(* PLC project TankLevelControl, PLCAutoPilot Tank Level Control 1.0 *)
(* stored: creationDateTime 2025-12-25T12:00:00, modificationDateTime 2025-12-25T12:00:00 *)

(* Dual Tank Level Control Program - Controls two pumps for tank filling - Pump 1: Fills Tank 1 from source - Pump 2: Transfers from Tank 1 to RO Tank - Includes start/stop, fault detection, and alarms *)
PROGRAM Tank_Control
  VAR
    System_Running : BOOL := FALSE;  (* System running flag *)
    Pump1_Cmd : BOOL := FALSE;  (* Pump 1 run command *)
    Pump2_Cmd : BOOL := FALSE;  (* Pump 2 run command *)
    Fault_Flag : BOOL := FALSE;  (* Fault active flag *)
    Pump1_Timer : TON;  (* Pump 1 delay timer *)
    Pump2_Timer : TON;  (* Pump 2 delay timer *)
  END_VAR
  VAR_INPUT
    LS_Tank1 : BOOL;  (* Tank 1 Level Switch (0=Low, 1=High) *)
    LS_RO_Tank : BOOL;  (* RO Tank Level Switch (0=Low, 1=High) *)
    PB_Start : BOOL;  (* Start Push Button (NO) *)
    PB_Stop : BOOL;  (* Stop Push Button (NC - TRUE when not pressed) *)
    PB_EStop : BOOL;  (* Emergency Stop (NC - TRUE when not pressed) *)
    OL_Pump1 : BOOL;  (* Pump 1 Overload (NC - TRUE when OK) *)
    OL_Pump2 : BOOL;  (* Pump 2 Overload (NC - TRUE when OK) *)
  END_VAR
  VAR_OUTPUT
    Pump1_Out : BOOL;  (* Pump 1 Output *)
    Pump2_Out : BOOL;  (* Pump 2 Output *)
    Running_Light : BOOL;  (* System Running Indicator *)
    Tank1_Low_Alarm : BOOL;  (* Tank 1 Low Level Alarm *)
    RO_Low_Alarm : BOOL;  (* RO Tank Low Level Alarm *)
    Fault_Light : BOOL;  (* Fault Indicator *)
  END_VAR

            
(* ================================================ *)
(* TANK LEVEL CONTROL PROGRAM                       *)
(* Dual Tank System with Pump Control               *)
(* Generated by PLCAutoPilot                        *)
(* ================================================ *)

(* ----- SYSTEM START/STOP LOGIC ----- *)
(* Start system when Start button pressed and safety OK *)
IF PB_Start AND PB_Stop AND PB_EStop AND NOT Fault_Flag THEN
    System_Running := TRUE;
END_IF;

(* Stop system when Stop button or E-Stop pressed *)
IF NOT PB_Stop OR NOT PB_EStop THEN
    System_Running := FALSE;
END_IF;

(* ----- FAULT DETECTION ----- *)
(* Set fault if any overload trips *)
IF NOT OL_Pump1 OR NOT OL_Pump2 THEN
    Fault_Flag := TRUE;
END_IF;

(* Reset fault when Start pressed and overloads OK *)
IF PB_Start AND OL_Pump1 AND OL_Pump2 THEN
    Fault_Flag := FALSE;
END_IF;

(* ----- PUMP 1 CONTROL (Fill Tank 1) ----- *)
(* Run Pump 1 when system running, Tank 1 is LOW, no fault *)
Pump1_Cmd := System_Running AND NOT LS_Tank1 AND OL_Pump1 AND NOT Fault_Flag;

(* Timer for Pump 1 start delay *)
Pump1_Timer(IN := Pump1_Cmd, PT := T#2S);

(* Pump 1 output with delay *)
Pump1_Out := Pump1_Timer.Q;

(* ----- PUMP 2 CONTROL (Fill RO Tank) ----- *)
(* Run Pump 2 when system running, RO Tank is LOW, Tank 1 is HIGH, no fault *)
Pump2_Cmd := System_Running AND NOT LS_RO_Tank AND LS_Tank1 AND OL_Pump2 AND NOT Fault_Flag;

(* Timer for Pump 2 start delay *)
Pump2_Timer(IN := Pump2_Cmd, PT := T#2S);

(* Pump 2 output with delay *)
Pump2_Out := Pump2_Timer.Q;

(* ----- INDICATOR OUTPUTS ----- *)
Running_Light := System_Running;
Tank1_Low_Alarm := System_Running AND NOT LS_Tank1;
RO_Low_Alarm := System_Running AND NOT LS_RO_Tank;
Fault_Light := Fault_Flag;
            
          
END_PROGRAM

FUNCTION_BLOCK GVL_IO
  VAR
    DI_Tank1_Level AT %IX0.0 : BOOL;  (* Tank 1 Level Switch Input *)
    DI_RO_Tank_Level AT %IX0.1 : BOOL;  (* RO Tank Level Switch Input *)
    DI_Start AT %IX0.2 : BOOL;  (* Start Button Input *)
    DI_Stop AT %IX0.3 : BOOL;  (* Stop Button Input *)
    DI_EStop AT %IX0.4 : BOOL;  (* Emergency Stop Input *)
    DI_OL_Pump1 AT %IX0.5 : BOOL;  (* Pump 1 Overload Input *)
    DI_OL_Pump2 AT %IX0.6 : BOOL;  (* Pump 2 Overload Input *)
    DO_Pump1 AT %QX0.0 : BOOL;  (* Pump 1 Output *)
    DO_Pump2 AT %QX0.1 : BOOL;  (* Pump 2 Output *)
    DO_Running AT %QX0.2 : BOOL;  (* Running Light Output *)
    DO_Tank1_Alarm AT %QX0.3 : BOOL;  (* Tank 1 Low Alarm Output *)
    DO_RO_Alarm AT %QX0.4 : BOOL;  (* RO Tank Low Alarm Output *)
    DO_Fault AT %QX0.5 : BOOL;  (* Fault Light Output *)
  END_VAR

            
(* I/O Mapping - This GVL maps physical I/O to symbolic names *)
            
          
END_FUNCTION_BLOCK

CONFIGURATION TankControl_Config
  RESOURCE TankControl_Resource ON PLC
    TASK MAST(INTERVAL := T#10ms, PRIORITY := 1);
    PROGRAM Tank_Control_Instance WITH MAST : Tank_Control;
  END_RESOURCE
END_CONFIGURATION
